// TIA Portal V20 export
DATA_BLOCK "test"   // DB145
// stored: Access Published, MemoryReserve 100, Namespace Unit1
   VAR
      "bool" : Array[0..19] of Bool;
      "int" : Array[0..19] of Int;
      "dint" : Array[0..19] of DInt;
      "real" : Array[0..19] of Real;
      Lreal : Array[0..19] of LReal;
      "Timer" : Array[0..19] of TON_TIME;
      Static_1 : USInt;
      Static_2 : USInt;
      Static_3 : USInt;
      bool_1 : Array[0..19] of Bool;
      ECH : Bool;
      CPM : LReal := 30.0;
   END_VAR
BEGIN
   // "bool"[19] : 모션 맵핑용 임시 변수
   // bool_1[19] : 모션 맵핑용 임시 변수
END_DATA_BLOCK
